DATA_BLOCK "KukaRobot1_CtrlDB"
{ S7_Optimized_Access := 'FALSE' }
VERSION : 0.1
// ATTRIBUTES
// AUTO_NUMBER = False
// BLOCK_NUMBER = 2401
// END_ATTRIBUTES
"KukaRobot1_Ctrl"

BEGIN

END_DATA_BLOCK

